(* CoDeSys 2.3.9.50 project: OneWire.pro *)
(* Libraries: TcBase.lib 14.5.09 12:14:08, TcSystem.lib 7.6.16 11:01:22, TcUtilities.lib 3.2.16 16:08:58, TcEtherCAT.lib 30.11.16 19:52:18, STANDARD.LIB 5.6.98 12:03:02, COMlibV2.lib 3.8.16 13:29:30 *)

(* Task configuration *)
TASK MAIN (PRIORITY := 0, INTERVAL := T#1ms);
	MAIN();
END_TASK

(* Global variable list: TwinCAT_Configuration *)
(* Generated automatically by TwinCAT - (read only) *)
VAR_CONFIG
	MAIN.serial_port_inputs AT %IB0 : EL6inData22B;
	MAIN.serial_port_outputs AT %QB0 : EL6outData22B;
END_VAR

(* Data type *)
TYPE E_Baudrate : (Baudrate4800, Baudrate9600);
END_TYPE

(* Data type *)
TYPE E_DataFrameFormat : (DataFrame8N1);
END_TYPE

(* Data type *)
TYPE E_OneWireResetResult : (WIRE_SHORTED, PRESENCE, ALARMING_PRESENCE, NO_PRESENCE);
END_TYPE

(* POU MAIN, ST *)
PROGRAM MAIN
VAR
	(* Serial Port Configuration *)
	serial_port_netid          : STRING := '5.32.119.18.3.1'; (* See "System Manager" -> "Gerät 2 (EtherCAT)" -> "EtherCAT" -> "NetId" *)
	serial_port_slave_address  : INT    := 1005;              (* See "System Manager" -> "Klemme 6 (EL6002)" -> "EtherCAT" -> "EtherCAT Adr" *)
	serial_port_coe_index      : UINT   := 16#8000;           (* 0x8000 for serial port 1, 0x8010 for serial port 2 *)

	(* 1-Wire Sensor Addresses *)
	temp_sensor_1_address : ARRAY[1..8] OF BYTE := 16#10, 16#38, 16#9E, 16#55, 16#03, 16#08, 16#00, 16#69; (* DS18S20 *)
	temp_sensor_2_address : ARRAY[1..8] OF BYTE := 16#10, 16#EF, 16#EF, 16#55, 16#03, 16#08, 16#00, 16#88; (* DS18S20 *)

	(* Temperatures *)
	temperature1 : REAL;
	temperature2 : REAL;

	(* 1-Wire *)
	OneWireAdapterReset       : OneWireAdapterReset;

	DS1820ConvertTemperature  : DS1820ConvertTemperature;
	DS1820ReadScratchPad      : DS1820ReadScratchPad;

	(* Serial Port *)
	serial_port_inputs  AT %I* : EL6inData22B;
	serial_port_outputs AT %Q* : EL6outData22B;

	SerialPortControl          : SerialLineControl;
	SerialPortRxBuffer         : ComBuffer;
	SerialPortTxBuffer         : ComBuffer;

	ClearComBuffer             : ClearComBuffer;

	(* State *)
	step : INT;

	lasterror : STRING(256);

	cycle_timer: TON;
END_VAR
SerialPortControl(Mode      := SERIALLINEMODE_EL6_22B,
                  pComIn    := ADR(serial_port_inputs),
                  pComOut   := ADR(serial_port_outputs),
                  SizeComIn := SIZEOF(serial_port_inputs),
                  RxBuffer  := SerialPortRxBuffer,
                  TxBuffer  := SerialPortTxBuffer);

CASE step OF
0: (* Init *)
	temperature1 := 0;
	temperature2 := 0;

	step := 100;

100: (* 1-Wire Adapter Reset / Initialization *)
	OneWireAdapterReset(EL6xNetId          := serial_port_netid,
                        EL6xSlaveAddr      := serial_port_slave_address,
                        EL6xCoEIndex       := serial_port_coe_index,
						SerialPortInputs   := serial_port_inputs,
                        SerialPortOutputs  := serial_port_outputs,
                        SerialPortRxBuffer := SerialPortRxBuffer,
                        SerialPortTxBuffer := SerialPortTxBuffer,
                        start              := FALSE);

	step := 200;

200:
	OneWireAdapterReset(SerialPortInputs   := serial_port_inputs,
                        SerialPortOutputs  := serial_port_outputs,
                        SerialPortRxBuffer := SerialPortRxBuffer,
                        SerialPortTxBuffer := SerialPortTxBuffer,
                        start              := TRUE);

	IF NOT OneWireAdapterReset.busy THEN
		IF OneWireAdapterReset.error THEN
			lasterror := CONCAT('1-Wire adapter reset failed. ', OneWireAdapterReset.errormsg);
			step := 0;
		ELSE
			step := 1000;
		END_IF
	END_IF

1000: (* Data Exchange Cycle *)
	cycle_timer(in := FALSE, pt := t#2.5s);
	cycle_timer(in := TRUE);

	(* Clear serial line communication buffer before each cycle in case synchronization has been lost... *)
    (* Tx- and Rx-Count should be zero after this point! *)
	ClearComBuffer(Buffer := SerialPortRxBuffer);
	ClearComBuffer(Buffer := SerialPortTxBuffer);

	step := 1050;

1050: (* Convert temperature *)
	DS1820ConvertTemperature(start := FALSE, rx := SerialPortRxBuffer, tx := SerialPortTxBuffer);

	step := 1100;

1100:
	DS1820ConvertTemperature(start := TRUE, rx := SerialPortRxBuffer, tx := SerialPortTxBuffer);

	IF NOT DS1820ConvertTemperature.busy THEN
		IF DS1820ConvertTemperature.error THEN
			lasterror := CONCAT('Temperature conversion failed. ', DS1820ConvertTemperature.errormsg);

			step := 0;
		ELSE
			step := 1200;
		END_IF
	END_IF

1200: (* Read temperature of sensor 1 *)
	DS1820ReadScratchPad(start   := FALSE,
                         address := temp_sensor_1_address,
                         rx      := SerialPortRxBuffer,
                         tx      := SerialPortTxBuffer);

	step := 1300;

1300:
	DS1820ReadScratchPad(start := TRUE,
                         rx    := SerialPortRxBuffer,
                         tx    := SerialPortTxBuffer);

	IF NOT DS1820ReadScratchPad.busy THEN
		IF DS1820ReadScratchPad.error THEN
			lasterror := CONCAT('Failed to exchange process data with temperature sensor 1. ', DS1820ReadScratchPad.errormsg);
			step := 0;
		ELSE
			temperature1 := DS1820ReadScratchPad.temperature;
			step := 1400;
		END_IF
	END_IF

1400: (* Read temperature of sensor 2 *)
	DS1820ReadScratchPad(start   := FALSE,
                         address := temp_sensor_2_address,
                         rx      := SerialPortRxBuffer,
                         tx      := SerialPortTxBuffer);

	step := 1500;

1500:
	DS1820ReadScratchPad(start := TRUE,
                         rx    := SerialPortRxBuffer,
                         tx    := SerialPortTxBuffer);

	IF NOT DS1820ReadScratchPad.busy THEN
		IF DS1820ReadScratchPad.error THEN
			lasterror := CONCAT('Failed to exchange process data with temperature sensor 2. ', DS1820ReadScratchPad.errormsg);
			step := 0;
		ELSE
			temperature2 := DS1820ReadScratchPad.temperature;
			step := 5000;
		END_IF
	END_IF

5000: (* Data Exchange Successful. Wait & repeat... *)
	cycle_timer(in := TRUE);

	IF cycle_timer.Q THEN
		step := 1000;
	END_IF
END_CASE
END_PROGRAM

(* POU OneWire/OneWireAdapterReset, ST *)
FUNCTION_BLOCK OneWireAdapterReset
(*
   Resets the 1-Wire adapter by first sending a 0x00 byte at 4800 bps,
   followed by a 0xC1 byte at 9600 bps for baud rate calibration.

   Finally resets the 1-wire bus for adapter presence detection.

   See DS2480B datasheet for details.
*)
VAR_INPUT
	start: BOOL;

	EL6xNetId: STRING;
	EL6xSlaveAddr: INT;
	EL6xCoEIndex: INT;
END_VAR
VAR_OUTPUT
	busy: BOOL;
	error: BOOL;
	errormsg: STRING;
END_VAR
VAR_IN_OUT
	SerialPortInputs   : EL6inData22B;
	SerialPortOutputs  : EL6outData22B;
	SerialPortRxBuffer : ComBuffer;
	SerialPortTxBuffer : ComBuffer;
END_VAR
VAR
	CoeWrite        : FB_EcCoESdoWrite;

	BAUDRATE_4800   : BYTE := 5;
	BAUDRATE_9600   : BYTE := 6;

	DATAFRAME_8N1   : BYTE := 3;

	TRUE_BYTE       : BYTE := 1;
	FALSE_BYTE      : BYTE := 0;

	SendByte        : SendByte;
	SerialLineReset : SerialLineReset;
	OneWireReset    : OneWireReset;

	step: INT;
	tmr: TON;
END_VAR
IF NOT start THEN
	step := 0;
END_IF

CASE step OF
0:
	IF start THEN
		busy := TRUE;
		error := FALSE;
		errormsg := '';

		CoeWrite.sNetId     := EL6xNetId;
		CoeWrite.nSlaveAddr := EL6xSlaveAddr;
		CoeWrite.nIndex     := EL6xCoEIndex;
		CoeWrite.tTimeout   := t#1s;

		step := 50;
	END_IF

50: (* Disable RTS/CTS *)
	CoeWrite.nSubIndex  := 16#01;
	CoeWrite.cbBufLen   := SIZEOF(FALSE_BYTE);
	CoeWrite.pSrcBuf    := ADR(FALSE_BYTE);

	CoeWrite(bExecute := FALSE);

	step := 51;

51:
	CoeWrite(bExecute := TRUE);

	IF NOT CoeWrite.bBusy THEN
		IF CoeWrite.bError THEN
			error := TRUE;
			errormsg := 'Disabling RTS/CTS failed.';

			step := 9999;
		ELSE
			step := 52;
		END_IF
	END_IF

52: (* Disable XON/XOFF on Tx Data *)
	CoeWrite.nSubIndex  := 16#02;
	CoeWrite.cbBufLen   := SIZEOF(FALSE_BYTE);
	CoeWrite.pSrcBuf    := ADR(FALSE_BYTE);

	CoeWrite(bExecute := FALSE);

	step := 53;

53:
	CoeWrite(bExecute := TRUE);

	IF NOT CoeWrite.bBusy THEN
		IF CoeWrite.bError THEN
			error := TRUE;
			errormsg := 'Disabling XON/XOFF on Tx Data failed.';

			step := 9999;
		ELSE
			step := 54;
		END_IF
	END_IF

54: (* Disable XON/XOFF on Rx Data *)
	CoeWrite.nSubIndex  := 16#03;
	CoeWrite.cbBufLen   := SIZEOF(FALSE_BYTE);
	CoeWrite.pSrcBuf    := ADR(FALSE_BYTE);

	CoeWrite(bExecute := FALSE);

	step := 55;

55:
	CoeWrite(bExecute := TRUE);

	IF NOT CoeWrite.bBusy THEN
		IF CoeWrite.bError THEN
			error := TRUE;
			errormsg := 'Disabling XON/XOFF on Rx Data failed.';

			step := 9999;
		ELSE
			step := 56;
		END_IF
	END_IF

56: (* Disable Send FIFO Data Continuous *)
	CoeWrite.nSubIndex  := 16#04;
	CoeWrite.cbBufLen   := SIZEOF(FALSE_BYTE);
	CoeWrite.pSrcBuf    := ADR(FALSE_BYTE);

	CoeWrite(bExecute := FALSE);

	step := 57;

57:
	CoeWrite(bExecute := TRUE);

	IF NOT CoeWrite.bBusy THEN
		IF CoeWrite.bError THEN
			error := TRUE;
			errormsg := 'Disabling continuous sending failed.';

			step := 9999;
		ELSE
			step := 58;
		END_IF
	END_IF

58: (* Disable Transfer Rate Optimization *)
	CoeWrite.nSubIndex  := 16#05;
	CoeWrite.cbBufLen   := SIZEOF(FALSE_BYTE);
	CoeWrite.pSrcBuf    := ADR(FALSE_BYTE);

	CoeWrite(bExecute := FALSE);

	step := 59;

59:
	CoeWrite(bExecute := TRUE);

	IF NOT CoeWrite.bBusy THEN
		IF CoeWrite.bError THEN
			error := TRUE;
			errormsg := 'Disabling transfer rate optimization failed.';

			step := 9999;
		ELSE
			step := 60;
		END_IF
	END_IF

60: (* Set data frame format to 8N1 *)
	CoeWrite.nSubIndex  := 16#15;
	CoeWrite.cbBufLen   := SIZEOF(DATAFRAME_8N1);
	CoeWrite.pSrcBuf    := ADR(DATAFRAME_8N1);

	CoeWrite(bExecute := FALSE);

	step := 61;

61:
	CoeWrite(bExecute := TRUE);

	IF NOT CoeWrite.bBusy THEN
		IF CoeWrite.bError THEN
			error := TRUE;
			errormsg := 'Setting data frame format to 8N1 failed.';

			step := 9999;
		ELSE
			step := 100;
		END_IF
	END_IF

100: (* Set baudrate to 4800bps *)
	CoeWrite.nSubIndex  := 16#11;
	CoeWrite.cbBufLen   := SIZEOF(BAUDRATE_4800);
	CoeWrite.pSrcBuf    := ADR(BAUDRATE_4800);

	CoeWrite(bExecute := FALSE);

	step := 200;

200:
	CoeWrite(bExecute := TRUE);

	IF NOT CoeWrite.bBusy THEN
		IF CoeWrite.bError THEN
			error := TRUE;
			errormsg := 'Setting baudrate to 4800bps failed.';

			step := 9999;
		ELSE
			step := 210;
		END_IF
	END_IF

210:
	tmr(in := FALSE, pt := t#100ms);

	step := 220;

220:
	tmr(in := TRUE);

	IF tmr.Q THEN
		step := 230;
	END_IF

230: (* Reset the serial port, clear buffers,... *)
	SerialLineReset(start     := FALSE,
	                pComIn    := ADR(SerialPortInputs),
	                pComOut   := ADR(SerialPortOutputs),
	                SizeComIn := SIZEOF(SerialPortInputs),
	                RxBuffer  := SerialPortRxBuffer,
	                TxBuffer  := SerialPortTxBuffer);
	step := 240;

240:
	SerialLineReset(start     := TRUE,
	                pComIn    := ADR(SerialPortInputs),
	                pComOut   := ADR(SerialPortOutputs),
	                SizeComIn := SIZEOF(SerialPortInputs),
	                RxBuffer  := SerialPortRxBuffer,
	                TxBuffer  := SerialPortTxBuffer);

	IF NOT SerialLineReset.busy THEN
		IF SerialLineReset.error THEN
			error := TRUE;
			errormsg := 'Serial line reset failed.';

			step := 9999;
		ELSE
			step := 300;
		END_IF
	END_IF

300: (* Send a null byte at 4800bps to initiate a master reset *)
	SendByte(SendByte := 16#00, TxBuffer := SerialPortTxBuffer);
	SendByte(SendByte := 16#00, TxBuffer := SerialPortTxBuffer);
	SendByte(SendByte := 16#00, TxBuffer := SerialPortTxBuffer);
	SendByte(SendByte := 16#00, TxBuffer := SerialPortTxBuffer);
	SendByte(SendByte := 16#00, TxBuffer := SerialPortTxBuffer);

	step := 400;

400: (* Wait until the null byte has been sent *)
	IF SerialPortTxBuffer.Count = 0 THEN
		step := 500;
	END_IF

500: (* Set baudrate back to 9600bps *)
	CoeWrite.nSubIndex  := 16#11;
	CoeWrite.cbBufLen   := SIZEOF(BAUDRATE_9600);
	CoeWrite.pSrcBuf    := ADR(BAUDRATE_9600);

	CoeWrite(bExecute := FALSE);

	step := 600;

600:
	CoeWrite(bExecute := TRUE);

	IF NOT CoeWrite.bBusy THEN
		IF CoeWrite.bError THEN
			error := TRUE;
			errormsg := 'Setting baudrate to 9600bps failed.';

			step := 9999;
		ELSE
			step := 610;
		END_IF
	END_IF

610: (* Reset the serial port, clear buffers,... *)
	SerialLineReset(start     := FALSE,
	                pComIn    := ADR(SerialPortInputs),
	                pComOut   := ADR(SerialPortOutputs),
	                SizeComIn := SIZEOF(SerialPortInputs),
	                RxBuffer  := SerialPortRxBuffer,
	                TxBuffer  := SerialPortTxBuffer);
	step := 620;

620:
	SerialLineReset(start     := TRUE,
	                pComIn    := ADR(SerialPortInputs),
	                pComOut   := ADR(SerialPortOutputs),
	                SizeComIn := SIZEOF(SerialPortInputs),
	                RxBuffer  := SerialPortRxBuffer,
	                TxBuffer  := SerialPortTxBuffer);

	IF NOT SerialLineReset.busy THEN
		IF SerialLineReset.error THEN
			error := TRUE;
			errormsg := 'Serial line reset failed.';

			step := 9999;
		ELSE
			step := 700;
		END_IF
	END_IF


700: (* First byte after reset must be a reset command for baud rate calibration *)
	SendByte(SendByte := 16#C1, TxBuffer := SerialPortTxBuffer);

	step := 750;

750: (* Wait until the calibration byte has been sent *)
	IF SerialPortTxBuffer.Count = 0 THEN
		step := 800;
	END_IF

800: (* Reset the serial port, clear buffers,... *)
	SerialLineReset(start     := FALSE,
	                pComIn    := ADR(SerialPortInputs),
	                pComOut   := ADR(SerialPortOutputs),
	                SizeComIn := SIZEOF(SerialPortInputs),
	                RxBuffer  := SerialPortRxBuffer,
	                TxBuffer  := SerialPortTxBuffer);
	step := 900;

900:
	SerialLineReset(start     := TRUE,
	                pComIn    := ADR(SerialPortInputs),
	                pComOut   := ADR(SerialPortOutputs),
	                SizeComIn := SIZEOF(SerialPortInputs),
	                RxBuffer  := SerialPortRxBuffer,
	                TxBuffer  := SerialPortTxBuffer);

	IF NOT SerialLineReset.busy THEN
		IF SerialLineReset.error THEN
			error := TRUE;
			errormsg := 'Serial line reset failed.';

			step := 9999;
		ELSE
			step := 1000;
		END_IF
	END_IF

1000: (* Check if a one wire reset works *)
	OneWireReset(start := FALSE, rx := SerialPortRxBuffer, tx := SerialPortTxBuffer);

	step := 1100;

1100:
	OneWireReset(start := TRUE, rx := SerialPortRxBuffer, tx := SerialPortTxBuffer);

	IF NOT OneWireReset.busy THEN
		IF OneWireReset.error OR OneWireReset.result = WIRE_SHORTED THEN
			error := TRUE;
			errormsg := '1-Wire reset failed.';

			step := 9999;
		ELSE
			step := 9999;
		END_IF
	END_IF

9999:
	busy := FALSE;
END_CASE
END_FUNCTION_BLOCK

(* POU OneWire/SerialLineReset, ST *)
FUNCTION_BLOCK SerialLineReset
(*
   Resets the serial port & clears all buffers.
*)
VAR_INPUT
	start: BOOL;
	pComIn: POINTER TO BYTE;
	pComOut: POINTER TO BYTE;
	SizeComIn: UINT;
END_VAR
VAR_OUTPUT
	busy: BOOL;
	error: BOOL;
	errormsg: STRING;
END_VAR
VAR_IN_OUT
	RxBuffer: ComBuffer;
	TxBuffer: ComBuffer;
END_VAR
VAR
	step: INT;

	ComReset: ComReset;
	ClearComBuffer: ClearComBuffer;
END_VAR
IF NOT start THEN
	step := 0;
END_IF

CASE step OF
0:
	IF start THEN
		busy := TRUE;
		error := FALSE;
		errormsg := '';

		step := 100;
	END_IF

100:
	ComReset(Execute := FALSE, pComIn := pComIn, pComOut := pComOut, SizeComIn := SizeComIn);

	step := 200;

200:
	ComReset(Execute := TRUE, pComIn := pComIn, pComOut := pComOut, SizeComIn := SizeComIn);

	IF NOT ComReset.Busy THEN
		IF ComReset.Error THEN
			error := TRUE;
			errormsg := 'ComReset failed.';
			step := 9999;
		ELSE
			step := 300;
		END_IF
	END_IF

300:
	ClearComBuffer(Buffer := RxBuffer);
	ClearComBuffer(Buffer := TxBuffer);

	step := 9999;

9999:
	busy := FALSE;
END_CASE
END_FUNCTION_BLOCK

(* POU OneWire/OneWireReset, ST *)
FUNCTION_BLOCK OneWireReset
(*
   Resets the 1-Wire bus.

   See DS2480B data sheet for details.
*)
VAR_INPUT
	start: BOOL;
END_VAR
VAR_OUTPUT
	busy: BOOL;
	error: BOOL;
	errormsg: STRING;

	result: E_OneWireResetResult;
END_VAR
VAR_IN_OUT
	rx: ComBuffer;
	tx: ComBuffer;
END_VAR
VAR
	step: INT;

	SendByte: SendByte;
	RecvByte: ReceiveByte;

	timeout: TON;
END_VAR
IF NOT start THEN
	step := 0;
END_IF

CASE step OF
0:
	IF start THEN
		busy := TRUE;
		error := FALSE;
		errormsg := '';

		timeout(in := FALSE, pt := t#1s);
		timeout(in := TRUE);

		SendByte(SendByte := 16#E3, TxBuffer := tx); (* Command Mode *)
		SendByte(SendByte := 16#C5, TxBuffer := tx); (* Reset Command, Speed=flex *)

		step := 100;
	END_IF

100:
	RecvByte(RxBuffer := rx);

	IF RecvByte.ByteReceived THEN
		IF (RecvByte.ReceivedByte AND 16#DC) = 16#CC THEN (* Reset Command Response *)
			CASE RecvByte.ReceivedByte AND 2#11 OF
				2#00: result := WIRE_SHORTED;
				2#01: result := PRESENCE;
				2#10: result := ALARMING_PRESENCE;
				2#11: result := NO_PRESENCE;
			ELSE
				error := TRUE;
				errormsg := 'Unknown reset state.';
			END_CASE
		ELSE
			error := TRUE;
			errormsg := 'Invalid reset response.';
		END_IF

		step := 9999;
	END_IF

	timeout(in := TRUE);

	IF timeout.Q THEN
		error := TRUE;
		errormsg := 'Timeout';

		step := 9999;
	END_IF

9999:
	busy := FALSE;
END_CASE
END_FUNCTION_BLOCK

(* POU OneWire/Sensors/DS1820ConvertTemperature, ST *)
FUNCTION_BLOCK DS1820ConvertTemperature
(*
   Makes all DS18S20 / DS18B20 sensors on the network start temperature conversion.

   See DS18S20 / DS18B20 data sheets for details.
*)
VAR_INPUT
	start: BOOL;
END_VAR
VAR_OUTPUT
	busy     : BOOL;
	error    : BOOL;
	errormsg : STRING;
END_VAR
VAR_IN_OUT
	rx: ComBuffer;
	tx: ComBuffer;
END_VAR
VAR
	step: INT;

	SendByte: SendByte;
	RecvByte: ReceiveByte;

	OneWireReset   : OneWireReset;
	OneWireSkipROM : OneWireSkipROM;

	timeout: TON;
END_VAR
IF NOT start THEN
	step := 0;
END_IF

CASE step OF
0:
	IF start THEN
		busy := TRUE;
		error := FALSE;
		errormsg := '';

		timeout(in := FALSE, pt := t#2.5s);
		timeout(in := TRUE);

		step := 100;
	END_IF

100:
	OneWireReset(start := FALSE, rx := rx, tx := tx);

	step := 200;

200:
	OneWireReset(start := TRUE, rx := rx, tx := tx);

	IF NOT OneWireReset.busy THEN
		IF OneWireReset.error THEN
			error := TRUE;
			errormsg := '1-Wire reset failed.';

			step := 9999;
		ELSE
			step := 300;
		END_IF
	END_IF

300:
	OneWireSkipROM(start := FALSE, rx := rx, tx := tx);

	step := 400;

400:
	OneWireSkipROM(start := TRUE, rx := rx, tx := tx);

	IF NOT OneWireSkipROM.busy THEN
		IF OneWireSkipROM.error THEN
			error := TRUE;
			errormsg := 'Skip ROM failed.';

			step := 9999;
		ELSE
			step := 500;
		END_IF
	END_IF

500:
	SendByte(SendByte := 16#E3, TxBuffer := tx); (* Set Command Mode *)
	SendByte(SendByte := 16#3B, TxBuffer := tx); (* Set Pullup Duration to 1048ms *)

	step := 600;

600:
	RecvByte(RxBuffer := rx);

	IF RecvByte.ByteReceived THEN
		IF RecvByte.ReceivedByte = 16#3A THEN (* Set Pullup Duration Response *)
			step := 700;
		ELSE
			error := TRUE;
			errormsg := 'Invalid set pull up duration response.';

			step := 9999;
		END_IF
	END_IF

	timeout(in := TRUE);

	IF timeout.Q THEN
		error := TRUE;
		errormsg := 'Timeout';

		step := 9999;
	END_IF

700:
	SendByte(SendByte := 16#EF, TxBuffer := tx); (* Arm 5V Strong Pullup *)
	SendByte(SendByte := 16#F1, TxBuffer := tx); (* Terminate Pulse - needed to save time. *)

	step := 800;

800:
	RecvByte(RxBuffer := rx);

	IF RecvByte.ByteReceived THEN
		IF (RecvByte.ReceivedByte AND 16#FC) = 16#EC THEN (* Arm 5V Strong Pullup Response *)
			step := 900;
		ELSE
			error := TRUE;
			errormsg := 'Invalid arm 5V strong pullup response.';

			step := 9999;
		END_IF
	END_IF

	timeout(in := TRUE);

	IF timeout.Q THEN
		error := TRUE;
		errormsg := 'Timeout';

		step := 9999;
	END_IF

900:
	SendByte(SendByte := 16#E1, TxBuffer := tx); (* Set Data Mode *)
	SendByte(SendByte := 16#44, TxBuffer := tx); (* Convert Temperature *)

	step := 1000;

1000:
	RecvByte(RxBuffer := rx);

	IF RecvByte.ByteReceived THEN
		IF RecvByte.ReceivedByte = 16#44 THEN (* Convert Temperature Response *)
			step := 1100;
		ELSE
			error := TRUE;
			errormsg := 'Invalid convert temperature response.';

			step := 9999;
		END_IF
	END_IF

	timeout(in := TRUE);

	IF timeout.Q THEN
		error := TRUE;
		errormsg := 'Timeout';

		step := 9999;
	END_IF

1100:
	RecvByte(RxBuffer := rx);

	IF RecvByte.ByteReceived THEN
		IF RecvByte.ReceivedByte = 16#76 OR RecvByte.ReceivedByte = 16#F6 THEN (* Pulse Response *)
			step := 1200;
		ELSE
			error := TRUE;
			errormsg := 'Invalid pulse response.';

			step := 9999;
		END_IF
	END_IF

	timeout(in := TRUE);

	IF timeout.Q THEN
		error := TRUE;
		errormsg := 'Timeout';

		step := 9999;
	END_IF

1200:
	SendByte(SendByte := 16#E3, TxBuffer := tx); (* Set Command Mode *)
	SendByte(SendByte := 16#ED, TxBuffer := tx); (* Disarm Strong Pullup *)
	SendByte(SendByte := 16#F1, TxBuffer := tx); (* Terminate Pulse - needed to save time. *)

	step := 1300;

1300:
	RecvByte(RxBuffer := rx);

	IF RecvByte.ByteReceived THEN
		IF (RecvByte.ReceivedByte AND 16#FC) = 16#EC THEN (* Disarm 5V Strong Pullup Response *)
			step := 9999;
		ELSE
			error := TRUE;
			errormsg := 'Invalid disarm strong pullup response.';

			step := 9999;
		END_IF
	END_IF

	timeout(in := TRUE);

	IF timeout.Q THEN
		error := TRUE;
		errormsg := 'Timeout';

		step := 9999;
	END_IF

9999:
	busy := FALSE;
END_CASE
END_FUNCTION_BLOCK

(* POU OneWire/OneWireSkipROM, ST *)
FUNCTION_BLOCK OneWireSkipROM
(*
   Selects all sensors on the 1-Wire network ("Skip ROM").

   See DS2480B data sheet for details.
*)
VAR_INPUT
	start: BOOL;
END_VAR
VAR_OUTPUT
	busy: BOOL;
	error: BOOL;
	errormsg: STRING;
END_VAR
VAR_IN_OUT
	rx: ComBuffer;
	tx: ComBuffer;
END_VAR
VAR
	step: INT;

	SendByte: SendByte;
	RecvByte: ReceiveByte;

	timeout: TON;
END_VAR
IF NOT start THEN
	step := 0;
END_IF

CASE step OF
0:
	IF start THEN
		busy := TRUE;
		error := FALSE;
		errormsg := '';

		timeout(in := FALSE, pt := t#1s);
		timeout(in := TRUE);

		SendByte(SendByte := 16#E1, TxBuffer := tx); (* Data Mode *)
		SendByte(SendByte := 16#CC, TxBuffer := tx); (* Skip ROM Command *)

		step := 100;
	END_IF

100:
	RecvByte(RxBuffer := rx);

	IF RecvByte.ByteReceived THEN
		IF RecvByte.ReceivedByte <> 16#CC THEN
			error := TRUE;
			errormsg := 'Invalid Skip ROM response.';
		END_IF

		step := 9999;
	END_IF

	timeout(in := TRUE);

	IF timeout.Q THEN
		error := TRUE;
		errormsg := 'Timeout';

		step := 9999;
	END_IF

9999:
	busy := FALSE;
END_CASE
END_FUNCTION_BLOCK

(* POU OneWire/Sensors/DS1820ReadScratchPad, ST *)
FUNCTION_BLOCK DS1820ReadScratchPad
(*
   Reads the "scratch pad" data from the selected temperature sensor,
   checks its CRC and calculates the temperature.

   See DS18S20 / DS18B20 data sheets for details.
*)
VAR_INPUT
	start: BOOL;

	address: ARRAY[1..8] OF BYTE;
END_VAR
VAR_OUTPUT
	busy     : BOOL;
	error    : BOOL;
	errormsg : STRING;

	scratchpad: ARRAY[1..9] OF BYTE;
	temperature: REAL;
END_VAR
VAR_IN_OUT
	rx: ComBuffer;
	tx: ComBuffer;
END_VAR
VAR
	step: INT;
	i: INT;

	max_tries : INT := 10;
	num_tries : INT;

	SendByte: SendByte;
	RecvByte: ReceiveByte;

	scratchpad_idx: INT;

	OneWireReset    : OneWireReset;
	OneWireMatchROM : OneWireMatchROM;
	OneWireCRC      : OneWireCRC;

	timeout: TON;
END_VAR
IF NOT start THEN
	step := 0;
END_IF

CASE step OF
0:
	IF start THEN
		busy     := TRUE;
		error    := FALSE;
		errormsg := '';

		num_tries := 0;

		step := 100;
	END_IF

100:
	timeout(in := FALSE, pt := t#500ms);
	timeout(in := TRUE);

	OneWireReset(start := FALSE, rx := rx, tx := tx);

	step := 200;

200:
	OneWireReset(start := TRUE, rx := rx, tx := tx);

	IF NOT OneWireReset.busy THEN
		IF OneWireReset.error THEN
			errormsg := CONCAT('1-Wire reset failed. ', OneWireReset.errormsg);
			step := 8000;
		ELSIF OneWireReset.result = NO_PRESENCE THEN
			errormsg := '1-Wire reset failed. No presence detected.';
			step := 8000;
		ELSIF OneWireReset.result = WIRE_SHORTED THEN
			errormsg := '1-Wire reset failed. Wire shorted.';
			step := 8000;
		ELSE
			step := 300;
		END_IF
	END_IF

300:
	OneWireMatchROM(start := FALSE, address := address, rx := rx, tx := tx);

	step := 400;

400:
	OneWireMatchROM(start := TRUE, rx := rx, tx := tx);

	IF NOT OneWireMatchROM.busy THEN
		IF OneWireMatchROM.error THEN
			errormsg := 'Match ROM failed.';

			step := 8000;
		ELSE
			step := 500;
		END_IF
	END_IF

500:
	SendByte(SendByte := 16#BE, TxBuffer := tx); (* Read Scratch Pad Command *)

	scratchpad_idx := 1;

	step := 600;

600:
	RecvByte(RxBuffer := rx);

	IF RecvByte.ByteReceived THEN
		IF RecvByte.ReceivedByte = 16#BE THEN (* Read Scratch Pad Command Response *)
			SendByte(SendByte := 16#FF, TxBuffer := tx); (* Send one byte to get one byte in response *)
			step := 700;
		ELSE
			errormsg := 'Invalid read scratch pad response.';

			step := 8000;
		END_IF
	END_IF

	timeout(in := TRUE);

	IF timeout.Q THEN
		errormsg := 'Timeout';

		step := 8000;
	END_IF

700:
	RecvByte(RxBuffer := rx);

	IF RecvByte.ByteReceived THEN
		scratchpad[scratchpad_idx] := RecvByte.ReceivedByte;

		scratchpad_idx := scratchpad_idx + 1;

		IF scratchpad_idx > SIZEOF(scratchpad) THEN
			step := 800;
		ELSE
			SendByte(SendByte := 16#FF, TxBuffer := tx); (* Send one byte to get one byte in response *)
		END_IF
	END_IF

	timeout(in := TRUE);

	IF timeout.Q THEN
		errormsg := 'Timeout';

		step := 8000;
	END_IF

800:
	OneWireCRC(pData := ADR(scratchpad), n := SIZEOF(scratchpad));

	IF OneWireCRC.crc <> 16#00 THEN
		errormsg := 'Invalid CRC.';

		step := 8000;
	ELSE
		step := 900;
	END_IF

900:
	CASE address[1] OF
	16#10: (* DS18S20 *)
		temperature := SHR(scratchpad[1], 1) - 0.25 + (scratchpad[8] - scratchpad[7]) / BYTE_TO_REAL(scratchpad[8]);

		IF temperature >= 85 THEN
			error := TRUE;
			errormsg := 'Invalid temperature.';
		END_IF
	16#28: (* DS18B20 *)
		temperature := (SHL(scratchpad[2], 8) + scratchpad[1]) / 16.0;

		IF temperature >= 85 THEN
			error := TRUE;
			errormsg := 'Invalid temperature.';
		END_IF
	ELSE
		error := TRUE;
		errormsg := 'Unknown sensor.';
	END_CASE

	step := 9999;

8000: (* Retry *)
	num_tries := num_tries + 1;

	IF num_tries >= max_tries THEN
		error := TRUE;
		step := 9999;
	ELSE
		step := 100;
	END_IF

9999:
	busy := FALSE;
END_CASE
END_FUNCTION_BLOCK

(* POU OneWire/OneWireMatchROM, ST *)
FUNCTION_BLOCK OneWireMatchROM
(*
   Selects a sensor on the 1-Wire network ("Match ROM").

   See DS2480B data sheet for details.
*)
VAR_INPUT
	start: BOOL;

	address: ARRAY[1..8] OF BYTE;
END_VAR
VAR_OUTPUT
	busy     : BOOL;
	error    : BOOL;
	errormsg : STRING;
END_VAR
VAR_IN_OUT
	rx: ComBuffer;
	tx: ComBuffer;
END_VAR
VAR
	step: INT;
	i: INT;
	countReceived: INT;

	SendByte: SendByte;
	RecvByte: ReceiveByte;

	timeout: TON;
END_VAR
IF NOT start THEN
	step := 0;
END_IF

CASE step OF
0:
	IF start THEN
		busy := TRUE;
		error := FALSE;
		errormsg := '';

		timeout(in := FALSE, pt := t#1s);
		timeout(in := TRUE);

		SendByte(SendByte := 16#E1, TxBuffer := tx); (* Data Mode *)
		SendByte(SendByte := 16#55, TxBuffer := tx); (* Match ROM Command *)

		FOR i := 1 TO SIZEOF(address) DO
			SendByte(SendByte := address[i], TxBuffer := tx);

			IF address[i] = 16#E3 THEN (* Byte 0xE3 must be escaped / sent twice *)
				SendByte(SendByte := address[i], TxBuffer := tx);
			END_IF
		END_FOR

		countReceived := 0;

		step := 100;
	END_IF

100:
	RecvByte(RxBuffer := rx);

	IF RecvByte.ByteReceived THEN
		IF RecvByte.ReceivedByte = 16#55 THEN
			step := 200;
		ELSE
			error := TRUE;
			errormsg := 'Invalid Match ROM response.';

			step := 9999;
		END_IF
	END_IF

	timeout(in := TRUE);

	IF timeout.Q THEN
		error := TRUE;
		errormsg := 'Timeout';

		step := 9999;
	END_IF

200:
	RecvByte(RxBuffer := rx);

	IF RecvByte.ByteReceived THEN
		countReceived := countReceived + 1;

		(* TODO Testen was passiert, wenn 0xE3 abgesendet wurde *)
		IF RecvByte.ReceivedByte <> address[countReceived] THEN
			error := TRUE;
			errormsg := 'Invalid response byte received.';

			step := 9999;
		ELSIF countReceived = SIZEOF(address) THEN
			step := 9999;
		END_IF
	END_IF

	timeout(in := TRUE);

	IF timeout.Q THEN
		error := TRUE;
		errormsg := 'Timeout';

		step := 9999;
	END_IF

9999:
	busy := FALSE;
END_CASE
END_FUNCTION_BLOCK

(* POU OneWire/OneWireCRC, ST *)
FUNCTION_BLOCK OneWireCRC
(*
   Plain 1-Wire CRC calculation...
*)
VAR_INPUT
	pData: UDINT;
	n: INT;
END_VAR
VAR_OUTPUT
	crc: BYTE;
END_VAR
VAR
	p: POINTER TO BYTE;
	i: INT;
END_VAR
VAR CONSTANT
	crctable: ARRAY[0..255] OF BYTE := 0, 94, 188, 226, 97, 63, 221, 131, 194, 156, 126, 32, 163, 253, 31, 65,
        157, 195, 33, 127, 252, 162, 64, 30, 95, 1, 227, 189, 62, 96, 130, 220,
        35, 125, 159, 193, 66, 28, 254, 160, 225, 191, 93, 3, 128, 222, 60, 98,
        190, 224, 2, 92, 223, 129, 99, 61, 124, 34, 192, 158, 29, 67, 161, 255,
        70, 24, 250, 164, 39, 121, 155, 197, 132, 218, 56, 102, 229, 187, 89, 7,
        219, 133, 103, 57, 186, 228, 6, 88, 25, 71, 165, 251, 120, 38, 196, 154,
        101, 59, 217, 135, 4, 90, 184, 230, 167, 249, 27, 69, 198, 152, 122, 36,
        248, 166, 68, 26, 153, 199, 37, 123, 58, 100, 134, 216, 91, 5, 231, 185,
        140, 210, 48, 110, 237, 179, 81, 15, 78, 16, 242, 172, 47, 113, 147, 205,
        17, 79, 173, 243, 112, 46, 204, 146, 211, 141, 111, 49, 178, 236, 14, 80,
        175, 241, 19, 77, 206, 144, 114, 44, 109, 51, 209, 143, 12, 82, 176, 238,
        50, 108, 142, 208, 83, 13, 239, 177, 240, 174, 76, 18, 145, 207, 45, 115,
        202, 148, 118, 40, 171, 245, 23, 73, 8, 86, 180, 234, 105, 55, 213, 139,
        87, 9, 235, 181, 54, 104, 138, 212, 149, 203, 41, 119, 244, 170, 72, 22,
        233, 183, 85, 11, 136, 214, 52, 106, 43, 117, 151, 201, 74, 20, 246, 168,
        116, 42, 200, 150, 21, 75, 169, 247, 182, 232, 10, 84, 215, 137, 107, 53;
END_VAR
crc := 0;

FOR i := 0 TO n-1 DO
	p := pData + i;
	crc := crctable[crc XOR p^];
END_FOR
END_FUNCTION_BLOCK
